TYPE EL5122_ENC_ControlChannel :
STRUCT
	{attribute addProperty Name "Control"}
	Control AT %Q* : EL5122_Control;
	{attribute addProperty Name "Set counter value"}
	SetCounterValue AT %Q* : UDINT;
END_STRUCT
END_TYPE

(* stored: Version 1.1.0.1, ProductVersion 3.1.4024.9
   DUT EL5122_ENC_ControlChannel: Id {33ad06e7-967c-0363-0683-65158144be3f} *)
